// TIA Portal V20 export
TYPE "PMC_Input_Data"
// stored: Access Published, Namespace CITI_Logic
   STRUCT
      Machining_Assembly : Struct
         FTQ_AllData_Rdy : Bool;
         FTQ_Data_Reset : Bool;
         Buffer_Bypass : Bool;
         Bypassed : Bool;
         CheckSum_OK : Bool;
         PUNData : String[20];
         FTQ_PUNData : String[20];
         GM_PartNumber : String[8];
         OptionalData : String[12];
         PartTypeString : String[12];
         FTQ_Reject_String : String[100];
         IncrGood_Count : Bool;
         IncrReject_Count : Bool;
         Machine_Loading : Bool;
         Machine_Unloading : Bool;
         Bypass_PartPallet_Inc : Bool;
         Part_Type : Int;
         Buffer_Count : Int;
         FTQ_Reject_Code : DInt;
         Material_Low : Bool;   // (See definition)
         AutoCycle_Running : Bool;
         ManualMode : Bool;
         Cycle_Time_Ready : Bool;
         OperatorOvercycle_1 : Bool;
         OperatorOvercycle_2 : Bool;
         Blocked : Bool;
         Starved : Bool;
         Idle : Bool;
         Wait_1 : Bool;
         Wait_2 : Bool;
         Wait_3 : Bool;
         Wait_4 : Bool;
         Stopped_by_Operator : Bool;
         Machine_Fault : Bool;
         Fault_Ack : Bool;
         Quality_Check_Warning : Bool;
         Quality_Check_Fault : Bool;
         Quality_Ack : Bool;
         ToolChange_Warning : Bool;
         ToolChange_Fault : Bool;
         ToolChange_Ack_Action : Bool;
         Andon_Hold : Bool;
         Fault_Word : DInt;
         Fault_String : String[200];
         Dry_Cycle_Mode : Bool;
         ControlPowerON : Bool;
         All_Maps_Out_Of_Auto : Bool;
         No_Maps_Show_Fault : Bool;
      END_STRUCT;
      Filter_Coolant : Struct
         Current_Temperature : Int;
         Numerical_Quan_1 : Int;
         Numerical_Quan_2 : Int;
         Numerical_Quan_3 : Int;
         Machine_Minor_Fault : Bool;
         Tank_Coolant_Temp_OK : Bool;
         Tank_Coolant_Temp_HI : Bool;
         Tank_Coolant_Temp_Low : Bool;
         Tank_Lvl_OK : Bool;
         Tank_Lvl_High : Bool;
         Tank_Lvl_Low : Bool;
         Pump_Back_Lvl_OK : Bool;
         Pump_Back_Lvl_High : Bool;
         Pump_Back_Lvl_Low : Bool;
      END_STRUCT;
      CMM : Struct
         Bad_Quality_Data : Bool;
         No_Queue_Avail : Bool;
         Queue_Avail : Bool;
         Insp_Prog_Running : Bool;
         Time_Remailing : Int;
      END_STRUCT;
   END_STRUCT;
END_TYPE
